(* CoDeSys 2.3 export: ADS_COMMUNICATION.EXP *)

(* POU ADS_Communication, CFC *)
PROGRAM ADS_Communication
VAR

	fb_floor1ADSwrite: ADSWRITE;
	fb_floor2ADSwrite: ADSWRITE;
	fb_floor4ADSwrite: ADSWRITE;

	heartbeat:TP;
END_VAR
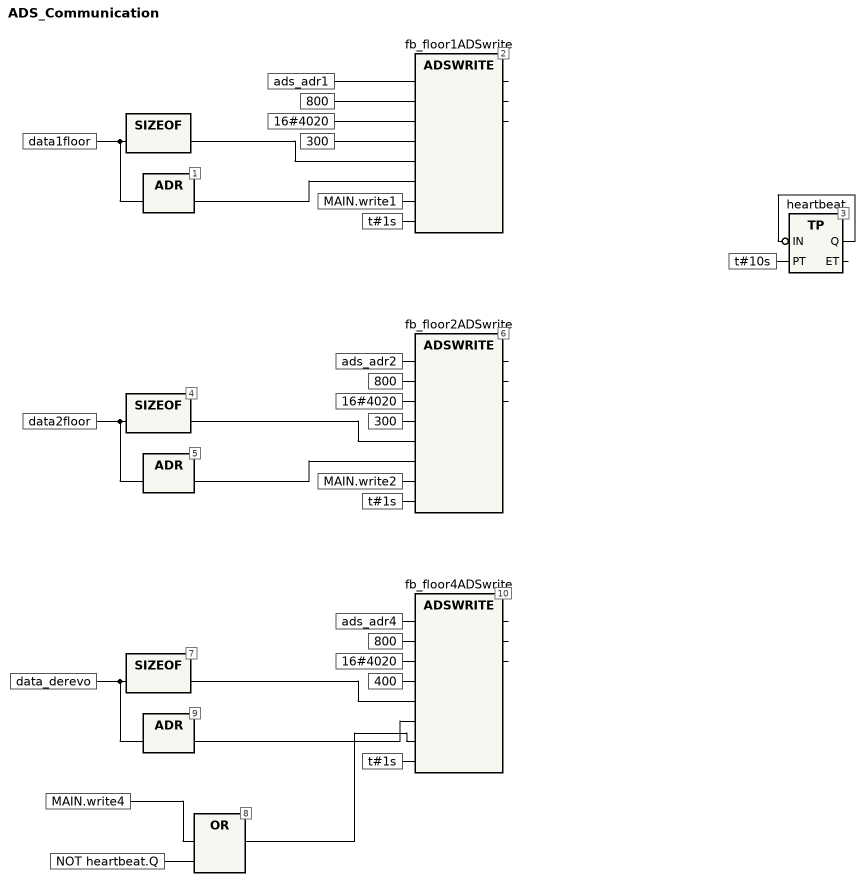
_CFC_ (* Continuous Function Chart, elements in execution order *)
#0 SIZEOF(data1floor)
#1 ADR(data1floor)
#2 fb_floor1ADSwrite:ADSWRITE(ads_adr1, 800, 16#4020, 300, #0, #1, MAIN.write1, t#1s)
#3 heartbeat:TP(IN: NOT #3.Q, PT: t#10s)
#4 SIZEOF(data2floor)
#5 ADR(data2floor)
#6 fb_floor2ADSwrite:ADSWRITE(ads_adr2, 800, 16#4020, 300, #4, #5, MAIN.write2, t#1s)
#7 SIZEOF(data_derevo)
#8 OR(MAIN.write4, NOT heartbeat.Q)
#9 ADR(data_derevo)
#10 fb_floor4ADSwrite:ADSWRITE(ads_adr4, 800, 16#4020, 400, #7, #9, #8, t#1s)
_END_CFC_
(* the same logic as Structured Text *)
fb_floor1ADSwrite(ads_adr1, 800, 16#4020, 300, SIZEOF(data1floor), ADR(data1floor), MAIN.write1, t#1s);
heartbeat(IN := NOT heartbeat.Q, PT := t#10s);
fb_floor2ADSwrite(ads_adr2, 800, 16#4020, 300, SIZEOF(data2floor), ADR(data2floor), MAIN.write2, t#1s);
fb_floor4ADSwrite(ads_adr4, 800, 16#4020, 400, SIZEOF(data_derevo), ADR(data_derevo), MAIN.write4 OR NOT heartbeat.Q, t#1s);
END_PROGRAM
